// TIA Portal V18 export
ORGANIZATION_BLOCK "Main"   // OB1, LAD, ProgramCycle
TITLE = "Main Program Sweep (Cycle)"
{ S7_Optimized_Access := 'TRUE' }
// stored: SetENOAutomatically false
   VAR_INPUT
      Initial_Call : Bool;   // Initial call of this OB
      Remanence : Bool;   // =True, if remanent data are available
   END_VAR
BEGIN

REGION Network 1
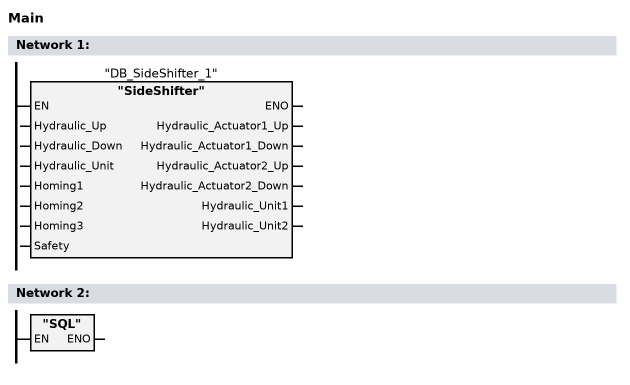
   RUNG wire#powerrail
      "DB_SideShifter_1"(Hydraulic_Up :=, Hydraulic_Down :=, Hydraulic_Unit :=, Homing1 :=, Homing2 :=, Homing3 :=, Safety :=, Hydraulic_Actuator1_Up =>, Hydraulic_Actuator1_Down =>, Hydraulic_Actuator2_Up =>, Hydraulic_Actuator2_Down =>, Hydraulic_Unit1 =>, Hydraulic_Unit2 =>)
   END_RUNG
   // the same network as SCL:
   "DB_SideShifter_1"();   // "SideShifter"
END_REGION

REGION Network 2
   RUNG wire#powerrail
      "SQL"()
   END_RUNG
   // the same network as SCL:
   "SQL"();
END_REGION
END_ORGANIZATION_BLOCK
